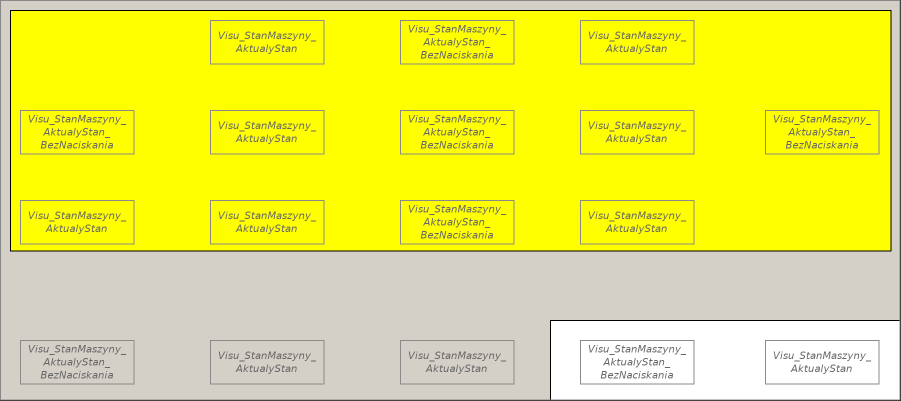
VISUALIZATION Visu_StanMaszyny_Diagram  // 901x401
VAR_IN_OUT
	
END_VAR
VAR_INPUT
	bWlaczPrzyciski								: BOOL;
END_VAR
    Rectangle (0,0 901x401)
    Rectangle (10,10 881x241)
    Frame (210,20 114x44), invisible if: not GVL_StanMaszyny.fbStanMaszyny.arrVisuTryb[GVL_StanMaszyny.fbStanMaszyny.iNumerTrybuPracy][12]
        shows Visu_StanMaszyny_AktualyStan(bNacisniety := GVL_StanMaszyny.fbStanMaszyny.bUnholdingZakonczone, stVisuStan := GVL_StanMaszyny.fbStanMaszyny.arrVisuStany [12])
    Frame (400,20 114x44), invisible if: not GVL_StanMaszyny.fbStanMaszyny.arrVisuTryb[GVL_StanMaszyny.fbStanMaszyny.iNumerTrybuPracy][11]
        shows Visu_StanMaszyny_AktualyStan_BezNaciskania(stVisuStan := GVL_StanMaszyny.fbStanMaszyny.arrVisuStany [11])
    Frame (580,20 114x44), invisible if: not GVL_StanMaszyny.fbStanMaszyny.arrVisuTryb[GVL_StanMaszyny.fbStanMaszyny.iNumerTrybuPracy][10]
        shows Visu_StanMaszyny_AktualyStan(bNacisniety := GVL_StanMaszyny.fbStanMaszyny.bHoldingZakonczone, stVisuStan := GVL_StanMaszyny.fbStanMaszyny.arrVisuStany [10])
    Frame (20,110 114x44), invisible if: not GVL_StanMaszyny.fbStanMaszyny.arrVisuTryb[GVL_StanMaszyny.fbStanMaszyny.iNumerTrybuPracy][4]
        shows Visu_StanMaszyny_AktualyStan_BezNaciskania(stVisuStan := GVL_StanMaszyny.fbStanMaszyny.arrVisuStany [4])
    Frame (210,110 114x44), invisible if: not GVL_StanMaszyny.fbStanMaszyny.arrVisuTryb[GVL_StanMaszyny.fbStanMaszyny.iNumerTrybuPracy][3]
        shows Visu_StanMaszyny_AktualyStan(bNacisniety := GVL_StanMaszyny.fbStanMaszyny.bStartingZakonczone, stVisuStan := GVL_StanMaszyny.fbStanMaszyny.arrVisuStany [3])
    Frame (400,110 114x44), invisible if: not GVL_StanMaszyny.fbStanMaszyny.arrVisuTryb[GVL_StanMaszyny.fbStanMaszyny.iNumerTrybuPracy][6]
        shows Visu_StanMaszyny_AktualyStan_BezNaciskania(stVisuStan := GVL_StanMaszyny.fbStanMaszyny.arrVisuStany [6])
    Frame (580,110 114x44), invisible if: not GVL_StanMaszyny.fbStanMaszyny.arrVisuTryb[GVL_StanMaszyny.fbStanMaszyny.iNumerTrybuPracy][16]
        shows Visu_StanMaszyny_AktualyStan(bNacisniety := GVL_StanMaszyny.fbStanMaszyny.bCompletingZakonczone, stVisuStan := GVL_StanMaszyny.fbStanMaszyny.arrVisuStany [16])
    Frame (765,110 114x44), invisible if: not GVL_StanMaszyny.fbStanMaszyny.arrVisuTryb[GVL_StanMaszyny.fbStanMaszyny.iNumerTrybuPracy][17]
        shows Visu_StanMaszyny_AktualyStan_BezNaciskania(stVisuStan := GVL_StanMaszyny.fbStanMaszyny.arrVisuStany [17])
    Frame (20,200 114x44), invisible if: not GVL_StanMaszyny.fbStanMaszyny.arrVisuTryb[GVL_StanMaszyny.fbStanMaszyny.iNumerTrybuPracy][15]
        shows Visu_StanMaszyny_AktualyStan(bNacisniety := GVL_StanMaszyny.fbStanMaszyny.bResetingSkonczone, stVisuStan := GVL_StanMaszyny.fbStanMaszyny.arrVisuStany [15])
    Frame (210,200 114x44), invisible if: not GVL_StanMaszyny.fbStanMaszyny.arrVisuTryb[GVL_StanMaszyny.fbStanMaszyny.iNumerTrybuPracy][14]
        shows Visu_StanMaszyny_AktualyStan(bNacisniety := GVL_StanMaszyny.fbStanMaszyny.bUnsuspendingZakonczone, stVisuStan := GVL_StanMaszyny.fbStanMaszyny.arrVisuStany [14])
    Frame (400,200 114x44), invisible if: not GVL_StanMaszyny.fbStanMaszyny.arrVisuTryb[GVL_StanMaszyny.fbStanMaszyny.iNumerTrybuPracy][5]
        shows Visu_StanMaszyny_AktualyStan_BezNaciskania(stVisuStan := GVL_StanMaszyny.fbStanMaszyny.arrVisuStany [5])
    Frame (580,200 114x44), invisible if: not GVL_StanMaszyny.fbStanMaszyny.arrVisuTryb[GVL_StanMaszyny.fbStanMaszyny.iNumerTrybuPracy][13]
        shows Visu_StanMaszyny_AktualyStan(bNacisniety := GVL_StanMaszyny.fbStanMaszyny.bSuspendingZakonczone, stVisuStan := GVL_StanMaszyny.fbStanMaszyny.arrVisuStany [13])
    Frame (20,340 114x44), invisible if: not GVL_StanMaszyny.fbStanMaszyny.arrVisuTryb[GVL_StanMaszyny.fbStanMaszyny.iNumerTrybuPracy][2]
        shows Visu_StanMaszyny_AktualyStan_BezNaciskania(stVisuStan := GVL_StanMaszyny.fbStanMaszyny.arrVisuStany [2])
    Frame (210,340 114x44), invisible if: not GVL_StanMaszyny.fbStanMaszyny.arrVisuTryb[GVL_StanMaszyny.fbStanMaszyny.iNumerTrybuPracy][7]
        shows Visu_StanMaszyny_AktualyStan(bNacisniety := GVL_StanMaszyny.fbStanMaszyny.bStoppingZakonczone, stVisuStan := GVL_StanMaszyny.fbStanMaszyny.arrVisuStany [7])
    Frame (400,340 114x44), invisible if: not GVL_StanMaszyny.fbStanMaszyny.arrVisuTryb[GVL_StanMaszyny.fbStanMaszyny.iNumerTrybuPracy][1]
        shows Visu_StanMaszyny_AktualyStan(bNacisniety := GVL_StanMaszyny.fbStanMaszyny.bClearingZakonczone, stVisuStan := GVL_StanMaszyny.fbStanMaszyny.arrVisuStany [1])
    Rectangle (550,320 351x81)
    Frame (580,340 114x44), invisible if: not GVL_StanMaszyny.fbStanMaszyny.arrVisuTryb[GVL_StanMaszyny.fbStanMaszyny.iNumerTrybuPracy][9]
        shows Visu_StanMaszyny_AktualyStan_BezNaciskania(stVisuStan := GVL_StanMaszyny.fbStanMaszyny.arrVisuStany [9])
    Frame (765,340 114x44), invisible if: not GVL_StanMaszyny.fbStanMaszyny.arrVisuTryb[GVL_StanMaszyny.fbStanMaszyny.iNumerTrybuPracy][8]
        shows Visu_StanMaszyny_AktualyStan(bNacisniety := GVL_StanMaszyny.fbStanMaszyny.bAbortingZakonczone, stVisuStan := GVL_StanMaszyny.fbStanMaszyny.arrVisuStany [8])
END_VISUALIZATION

(* stored: Version 1.1.0.1, ProductVersion 3.1.4024.11
   Visu Visu_StanMaszyny_Diagram: Id {deb2aa69-5bd6-4629-931b-818c74178be8} *)
